FUNCTION_BLOCK FB_SafetySignalsAK
VAR_INPUT
	SZPCo			: BOOL; //Safety Zone Pallet Conveyor 1	
	//NrOfContactor 	: INT :=3;//Number of contactors in cabinet
END_VAR
VAR_OUTPUT
END_VAR
VAR_IN_OUT
	SGref			: FB_ProBOXSG; //Reference to Switching group
	AKSignals		: ST_ProBoxSafetyAK;
END_VAR
VAR
	//fbBlink_1s	: FB_GeneratePulse := (Start := TRUE, PulseTimeOn := T#1S, PulseTimeOff := T#1S); // Blink 1s
	i,iMax		: INT;
	EmgStatus	: ST_EmgStatus;
END_VAR

//check if ResetSafetyNeeded
EmgStatus.eExternal := SZPCo;
EmgStatus.eInternal := AKSignals.Inputs.EsOk;
EmgStatus.eInternError := (AKSignals.Inputs.ComErr OR AKSignals.Inputs.FBErr); 
SGref.M_SetEmgStatus(EmgStatus);

//Pass signals from input to output
AKSignals.Outputs.ContactorOn 	:= SGref.CtrlOut.OpSummary.OpMcOn;
AKSignals.Outputs.ContactorOff 	:= SGref.CtrlOut.OpSummary.OpMcOff;
AKSignals.Outputs.ErrorAck 		:= SGref.CtrlOut.OpSummary.OpResetSafety;

// Copy over all feedback signals from SG group to be transfered to Safety							   
MEMCPY(ADR(AKSignals.Outputs.FeedBackContactor),ADR(SGref.HW_Inputs.Diag.FeedbackMainContactorOFF),SIZEOF(AKSignals.Outputs.FeedBackContactor));

END_FUNCTION_BLOCK

(* stored: Version 1.1.0.1, ProductVersion 3.1.4024.9
   POU FB_SafetySignalsAK: Id {7d24fa79-6de6-4756-9d0e-a20d60c800e3}, SpecialFunc None *)
